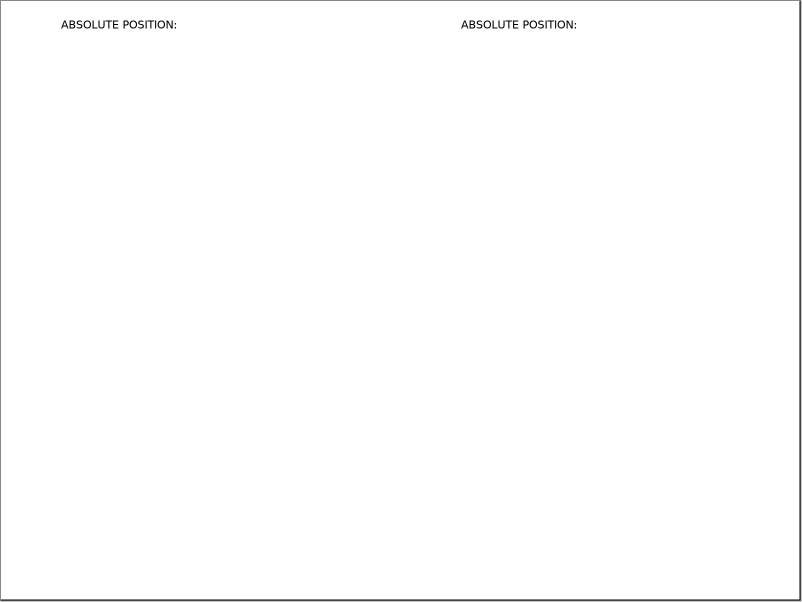
VISUALIZATION F31_Move_Superimposed  // 802x602
    Rectangle (0,0 800x600)
    Label (10,10 170x30), "ABSOLUTE POSITION:"
    Label (410,10 170x30), "ABSOLUTE POSITION:"
END_VISUALIZATION

(* stored: Version 1.1.0.1, ProductVersion 3.1.4022.7
   Visu F31_Move_Superimposed: Id {f799719c-4492-41fe-909c-680e55acea2b} *)
